// TIA Portal V18 export
ORGANIZATION_BLOCK "Main"   // OB1, LAD, ProgramCycle
TITLE = "Main Program Sweep (Cycle)"
{ S7_Optimized_Access := 'TRUE' }
VERSION : 0.1
// stored: AutoNumber true, IsIECCheckEnabled false, SetENOAutomatically false
   VAR_INPUT
      Initial_Call : Bool;   // Initial call of this OB
      Remanence : Bool;   // =True, if remanent data are available
   END_VAR
   VAR_TEMP
      qqq : Bool;
      qqqqq : Bool;
   END_VAR
BEGIN

REGION Network 1
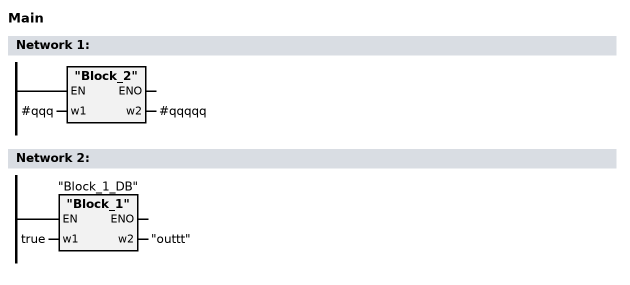
   RUNG wire#powerrail
      "Block_2"(w1 := #qqq, w2 => #qqqqq)
   END_RUNG
   // the same network as SCL:
   "Block_2"(w1 := #qqq, w2 => #qqqqq);
END_REGION

REGION Network 2
   RUNG wire#powerrail
      "Block_1_DB"(w1 := true, w2 => "outtt")
   END_RUNG
   // the same network as SCL:
   "Block_1_DB"(w1 := true, w2 => "outtt");   // "Block_1"
END_REGION
END_ORGANIZATION_BLOCK
